TYPE St_DefaultIdentity :
STRUCT
	SKU					:STRING;
	GTIN				:STRING;
	ProductionOrder		:STRING;
	LocalProductionOrder:STRING;
	PITCode				:STRING;
	BatchID				:STRING;
	ProductionLine		:STRING;
END_STRUCT
END_TYPE

(* stored: Version 1.1.0.1, ProductVersion 3.1.4024.13
   DUT St_DefaultIdentity: Id {baf42b41-2fbf-4886-a2ee-203d05dabc47} *)
